{attribute 'GeneratedUsingTerminal: APS1003-7000-0016'}
{attribute addProperty BoxType "APS1003-7000-0016"}
{attribute addProperty Id "EtcSlaveTerminalBaseYVR_InputsAT %I*YVR_Inputs_4719D0DB98YVR_OutputsAT %Q*YVR_Outputs_31F2CBB3146WcStateAT %I*WcState_9091E0EB2InfoDataAT %I*InfoData_BEF6B88E18"}
{attribute addProperty CRC "2154999165"}
{attribute addProperty Size "264"}
TYPE APS1003_8072AD7D EXTENDS EtcSlaveTerminalBase :
STRUCT
	{attribute addProperty Name "YVR_Inputs"}
	YVR_Inputs : YVR_Inputs_4719D0DB;
	{attribute addProperty Name "YVR_Outputs"}
	YVR_Outputs : YVR_Outputs_31F2CBB3;
	{attribute addProperty Name "WcState"}
	WcState : WcState_9091E0EB;
	{attribute addProperty Name "InfoData"}
	InfoData : InfoData_BEF6B88E;
END_STRUCT
END_TYPE

(* stored: Version 1.2.0.0, ProductVersion 3.1.4024.9
   DUT APS1003_8072AD7D: Id {872cb7c7-3c7b-4ead-b295-66c01052544d} *)
